TYPE TFRulliera_IN :
STRUCT
	
	FTC_Presenza1 			: BOOL; // Fotocellula Presenza 1 "INGRESSO"
	FTC_Presenza1Enable 	: BOOL; // Fotocellula Presenza 1 Abilitata
	
	FTC_Presenza2		 	: BOOL; // Fotocellula Presenza 2 "MEDIANA"
	FTC_Presenza2Enable 	: BOOL; // Fotocellula Presenza 2 Abilitata 
	
	FTC_Presenza3		 	: BOOL; // Fotocellula Presenza 3 "USCITA"
	FTC_Presenza3Enable		: BOOL; // Fotocellula Presenza 3 Abilitata 
	
END_STRUCT
END_TYPE

(* stored: Version 1.1.0.1, ProductVersion 3.1.4024.11
   DUT TFRulliera_IN: Id {820cfcf8-0f8e-4385-8168-73bae4ad58c2} *)
